// TIA Portal V16 export
// export: Created 2023-03-29T11:04:55.8606316Z, ExportSetting WithDefaults, DisplayName Totally Integrated Automation Portal, DisplayVersion V16 Update 6, DisplayName TIA Portal Version Control Interface, DisplayVersion V16 Update 2, DisplayName TIA Portal Openness, DisplayVersion V16 Update 6, DisplayName STEP 7 Professional, DisplayVersion V16 Update 6, DisplayName STEP 7 Safety, DisplayVersion V16, DisplayName WinCC Advanced, DisplayVersion V16 Update 6
DATA_BLOCK "Write_dbHold_TCP_Sending_DB"   // DB112
VERSION : 0.1
// stored: AutoNumber true, DBAccessibleFromOPCUA true, InstanceOfName Write_dbHold_TCP_Sending, InstanceOfType FB
"Write_dbHold_TCP_Sending"
BEGIN
END_DATA_BLOCK
